TYPE ST_BaseHMIConnectorEvents_DetailInformation :
STRUCT
	uiIDEvent						: UINT;
	uiIDItem						: UINT;				//id elementu
	sCode							: STRING;			//kod elementu
	bActive							: BOOL;
	bIgnoreRepetitions				: BOOL;				//jak true nie zliczaj powtorzeń wystapienia np komunikaty
	uiRepetitionCounter				: UINT;
	sStart							: STRING;			//poczatek wystepowania zgłoszenia
	sFinish							: STRING;			//koniec wystepowaniazgloszenia
	sConfirmed						: STRING;			// stempel potwierdzenia 
	bConfirm						: BOOL;				//informacja czy potrzebne jest potwierdzenie 
	bConfirmed						: BOOL;				//pamięta czy już potwierdzone
	sEventCategory					: STRING;
	wsDescription					: WSTRING;
	wsDescriptionFull				: WSTRING;
END_STRUCT
END_TYPE

(* stored: Version 1.1.0.1
   DUT ST_BaseHMIConnectorEvents_DetailInformation: Id {e8441c86-f5c1-0299-2525-2b849bd64d99} *)
